TYPE ControllerParameters :
STRUCT
	PV: LREAL;
	SP: LREAL; // $(write 0, setup, read 0, decimals 1, step 0.5)
	SP_HighSpeed: LREAL;
	CSP: LREAL;	// Beräknat börvärde
	P: LREAL := 2; // $(write 1, setup, read 0, decimals 3, step 0.001)
	I: TIME := T#2M; // $(write 1, setup, read 0, time "m:s")
	D: TIME := T#10m; // $(write 1, setup, read 0, time "m:s")
	CV: LREAL;
END_STRUCT
END_TYPE

(* stored: Version 1.1.0.1, ProductVersion 3.1.4024.6
   DUT ControllerParameters: Id {5d6aeccb-a356-4f0c-a7b2-32ace91878aa} *)
